// Mitsubishi GX Works2 project: 0625(Off Delay,펄스타이머)   PLC: Q02/Q02H

PROGRAM MAIN
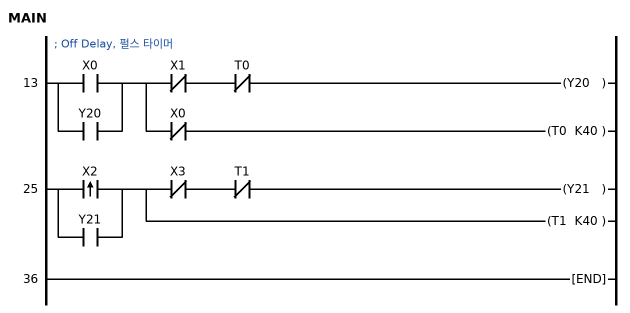
; Off Delay, 펄스 타이머
13    LD      X0
      OR      Y20
      MPS
      ANI     X1
      ANI     T0
      OUT     Y20
      MPP
      ANI     X0
      OUT     T0 K40
25    LDP     X2
      OR      Y21
      MPS
      ANI     X3
      ANI     T1
      OUT     Y21
      MPP
      OUT     T1 K40
36    END
END_PROGRAM
